(* CoDeSys 2.3.9.50 project: 2C.pr6 *)
(* Libraries: STANDARD.LB6 5.6.98 12:03:02 *)

(* POU MAIN, LD *)
PROGRAM MAIN
VAR
	Aoff AT %IX0.1: BOOL;
	A AT %IX0.0: BOOL;
	Boff AT %IX0.1: BOOL;
	B AT %IX0.2: BOOL;
	Coff AT %IX0.1: BOOL;
	C AT %IX0.3: BOOL;
	Doff AT %IX0.1: BOOL;
	D AT %IX0.4: BOOL;
	InterlockA AT %IX0.5: BOOL;
	InterlockB AT %IX0.6: BOOL;
	Fan AT %QX0.0: BOOL;
END_VAR
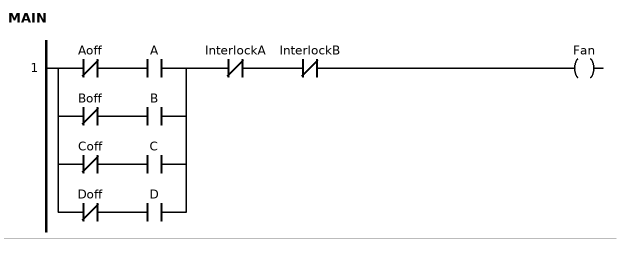
_LD_ (* Ladder Diagram *)
NETWORK 1
	{ [/Aoff] - [A] | [/Boff] - [B] | [/Coff] - [C] | [/Doff] - [D] } - [/InterlockA] - [/InterlockB] --- (Fan)
_END_LD_
(* the same logic as Structured Text *)
(* Network 1 *)
Fan := (NOT Aoff AND A OR NOT Boff AND B OR NOT Coff AND C OR NOT Doff AND D) AND NOT InterlockA AND NOT InterlockB;
END_PROGRAM

(* Visualisation Q2C
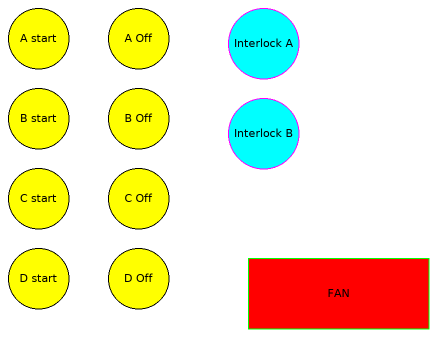
ellipse at (60,50)-(121,111): text "A start"; alarm colour if %IX0.0; toggles %IX0.0
ellipse at (60,210)-(121,271): text "C start"; alarm colour if %IX0.3; toggles %IX0.3
ellipse at (60,130)-(121,191): text "B start"; alarm colour if %IX0.2; toggles %IX0.2
ellipse at (60,290)-(121,351): text "D start"; alarm colour if %IX0.4; toggles %IX0.4
ellipse at (160,50)-(221,111): text "A Off"; alarm colour if %IX0.1; toggles %IX0.1
ellipse at (160,130)-(221,191): text "B Off"; alarm colour if %IX0.1; toggles %IX0.1
ellipse at (160,210)-(221,271): text "C Off"; alarm colour if %IX0.1; toggles %IX0.1
ellipse at (160,290)-(221,351): text "D Off"; alarm colour if %IX0.1; toggles %IX0.1
ellipse at (280,50)-(351,121): text "Interlock A"; alarm colour if %IX0.5; toggles %IX0.5
ellipse at (280,140)-(351,211): text "Interlock B"; alarm colour if %IX0.6; toggles %IX0.6
rectangle at (300,300)-(481,371): text "FAN"; alarm colour if %QX0.0
*)
